(* Logix 5000 project; controller DispersionPlc vendor 1 type 14 code 108 rev 34.11; software revision 34.01; part 6 of 22 *)
(* tags used below, declared in another part *)
   D_AlarmTimers : TIMER[200];
   D_AlarmTimers2 : TIMER[100];
   Disp_AlarmScanIdx : DINT;
   Disp_NewAlarmScanIdx : DINT;
   DispAlarmDisplayTmr : TIMER;
   DispersionAckAlarms : BOOL[128];
   DPT_4320_Holding : REAL;
   DPT_4320_Samples : DINT;
   InxTog : BOOL[32];
   NoNEwAlarmsDestedted : BOOL;
   ONS : BOOL[32];
   _Placeholder : DINT;
   AFB : BOOL;
   AFI : BOOL;
   AG4302_LLP_Alarm : BOOL;
   B4320_PumpAutoCommand : BOOL;
   B4320_PumpManCommand : BOOL;
   B4320_PumpManStart : AOI_Toggle;
   Both_Running : BOOL;
   Both_Running_Timer : TIMER;
   Cat_Destination_K400 : BOOL;
   Cat_Destination_T4301 : BOOL;
   Cat_Tank_Destination : DINT;
   Disp_AlarmsResetting : BOOL;
   Disp_Alr_To_Sound_Horn : BOOL[128];
   Disp_AlrResetIdx : DINT;
   Disp_QuedAlarm : DINT;
   DispAlarmResetBit : BOOL;
   DispersionAlarms : BOOL[256];
   DPT_4320 : REAL;
   DPT_4320_FILL : REAL;
   DPT_4320_Holding1 : REAL;
   DPT_4320_OffSet : REAL;
   DPT_4320_Raw : INT;
   DPT_4320_Sf : REAL;
   dpthighraw : REAL;
   dptlowraw : REAL;
   Drum_Transfer : BOOL;
   Emergency_Cool_4301 : BOOL;
   Enable_High_Alarm : BOOL;
   Estop_Inx : ALIAS FOR Local:3:I.Data.3;
   EstopBulk_upper : ALIAS FOR Local:1:O.Data[27].15;
   FE_4303 : REAL;
   FE_4303_Low : REAL;
   FE_4304 : REAL;
   FE_4304_Low : REAL;
   HMI_Linked_Timer : REAL;
   Hold_For_Flow_Switch : BOOL;
   HornONS_Phases : BOOL[32];
   HS_9A249 : ALIAS FOR Local:1:O.Data[0].17;
   HS_9A640 : ALIAS FOR Local:1:O.Data[0].18;
   InxAlarms : BOOL[128];
   K4_High_Temp : BOOL;
   K4_Low_Temp : BOOL;
   Linked_Timer : TIMER;
   LS_4302_High : BOOL;
   MCC1D4_20_TT5_Relay : BOOL;
   MCC1F3_TT1_Relay : BOOL;
   MCC1F4_8_TT9_Relay : BOOL;
   Melamine_Amount_Per_Count : REAL;
   Melamine_Charge_Remaining : REAL;
   Melamine_Flow_Rate : REAL;
   Melamine_Flow_Raw : INT;
   Melamine_Flow_Raw_Adjusted : REAL;
   Melamine_Flow_Scale_Factor : REAL;
   Melamine_Last_Charge : REAL;
   Melamine_Manual_Start : BOOL;
   Melamine_Pump_Off : BOOL;
   Melamine_Pump_Run : BOOL;
   Melamine_Transfer : BOOL;
   Melamine_transfer_amount : REAL;
   melamine_transfer_setpoint : REAL;
   MelaminePumpTmr : TIMER;
   Melimine_Max_Flow : DINT;
   Melimine_Pump_Manual_Run : BOOL;
   MIXER_A_4320_RUN : ALIAS FOR Local:1:O.Data[0].5;
   MMI_A_4320_RUN_PB : BOOL;
   MMI_Disp_Alarm_Reset_Pb : BOOL;
   MMI_INX_Solvent_Bypass : BOOL;
   MMI_INX_Solvent_Bypass_TOG : BOOL;
   MMI_P_4303_Run_Pb : BOOL;
   MMI_P_4304_RUN_PB : BOOL;
   MMI_P_4320_RUN_PB : BOOL;
   MMI_XV_4320_1_PB : BOOL;
   MMI_XV_4320_2_PB : BOOL;
   Mon_Destination_K400 : BOOL;
   Mon_Destination_T4301 : BOOL;
   Mon_Tank_Destination : DINT;
   NM_4303_AOI : AStd_AI_AOI;
   NM_4303_O2 : AStd_AnalogInput;
   O7_10_BUZ : ALIAS FOR Local:7:O.Data.10;
   One_Shots : DINT;
   OneShots : DINT;
   ONSTog : DINT;
   Phase_AlarmHorn : BOOL;
   Pv_Disp_Alarm_Val : DINT;
   RG_T52_AI_Raw : INT;
   RG_T53_AI_Raw : INT;
   RTA_Input_Floats : REAL[100];
   SPARE_I_1_4_5 : ALIAS FOR Local:1:I.Data[4].5;
   SPARE_O_1_0_21 : ALIAS FOR Local:1:O.Data[0].21;
   ST_K400_1 : REAL;
   ST_K400_1_LOW : REAL;
   ST_K400_1_Timer : TIMER[6];
   ST_K400_SAFETY : BOOL;
   Start_Melamine_Transfer_PB : BOOL;
   T4301_AIR_PURGE_REQUEST : BOOL;
   T4301_Cooling_On : BOOL;
   T4301_Heating_On : BOOL;
   T4301_K : Kettle;
   T4301_Mixer : VFD;
   T4301_Process_Alarm_Setpoints : Alarm_SPT;
   T4301_Temp_Feed_Alarm : DINT;
   T4302_Cooling_Pressure : DINT;
   T4302_Cooling_Pressure_SPT : DINT;
   T4302_DISCHARGE : BOOL;
   t4302_Line_pressure_High : BOOL;
   t4302_Line_pressure_Hightmr : TIMER;
   T53_Mixer : VFD;
   Tank_Link_Enable : BOOL;
   Tank_Link_Enable_ONS : BOOL;
   Tank_Link_Enable_ONS1 : BOOL;
   Tank_Link_ONS : BOOL[32];
   Tank_Linked : BOOL;
   TE_4301A : ALIAS FOR Local:8:I.Ch0Data;
   Te_4301A_High : REAL;
   TE_4301A_Low : REAL;
   TE_4320 : INT;
   TIT_S51_1 : AStd_AnalogInput;
   TOGGLE : BOOL;
   TRANS_PUMP_P_4320_RUN : ALIAS FOR Local:1:O.Data[0].6;
   TransferDone : BOOL;
   TruckLoadLevelAlarmResetPBLight : BOOL;
   V4304_Pump : VFD;
   Vaild_Monomer_Barcode : BOOL;
   VFD_4302_1 : AStd_VFD;
   W4303_Pump : VFD;
   WIT_4302_1 : AStd_AnalogInput;
   WIT_4306_1 : AStd_AnalogInput;
   WIT_4307_1 : AStd_AnalogInput;
   XI_K400_1 : BOOL;
   XV_4303_01 : ALIAS FOR Local:5:O.Data.3;
   XV_4303_03 : BOOL;
   XV_4303_04 : BOOL;
   XV_4303_05 : BOOL;
   XV_4304 : ALIAS FOR Local:5:O.Data.4;
   XV_4304_02 : BOOL;
   XV_4304_03 : BOOL;
   XV_4304_04 : BOOL;
   XV_4320_1 : ALIAS FOR Local:1:O.Data[1].1;
   XV_4320_2 : ALIAS FOR Local:1:O.Data[1].0;
   XV_K400_03_SEQCLOSE : BOOL;
   XV_K400_04_SEQCLOSE : BOOL;
   ZSC_4303_03 : BOOL;
   ZSC_4303_04 : BOOL;
   ZSC_4303_05 : BOOL;
   ZSC_4304_02 : BOOL;
   ZSC_4304_03 : BOOL;
   ZSC_4304_04 : BOOL;
   ZSC_4320_1 : ALIAS FOR Local:1:I.Data[4].3;
   ZSO_4303_03 : BOOL;
   ZSO_4303_04 : BOOL;
   ZSO_4303_05 : BOOL;
   ZSO_4304_02 : BOOL;
   ZSO_4304_03 : BOOL;
   ZSO_4304_04 : BOOL;
   ZSO_4320_1 : ALIAS FOR Local:1:I.Data[4].2;
   ZSO_4320_2 : ALIAS FOR Local:1:I.Data[4].0;
(* MainProgram, continued *)

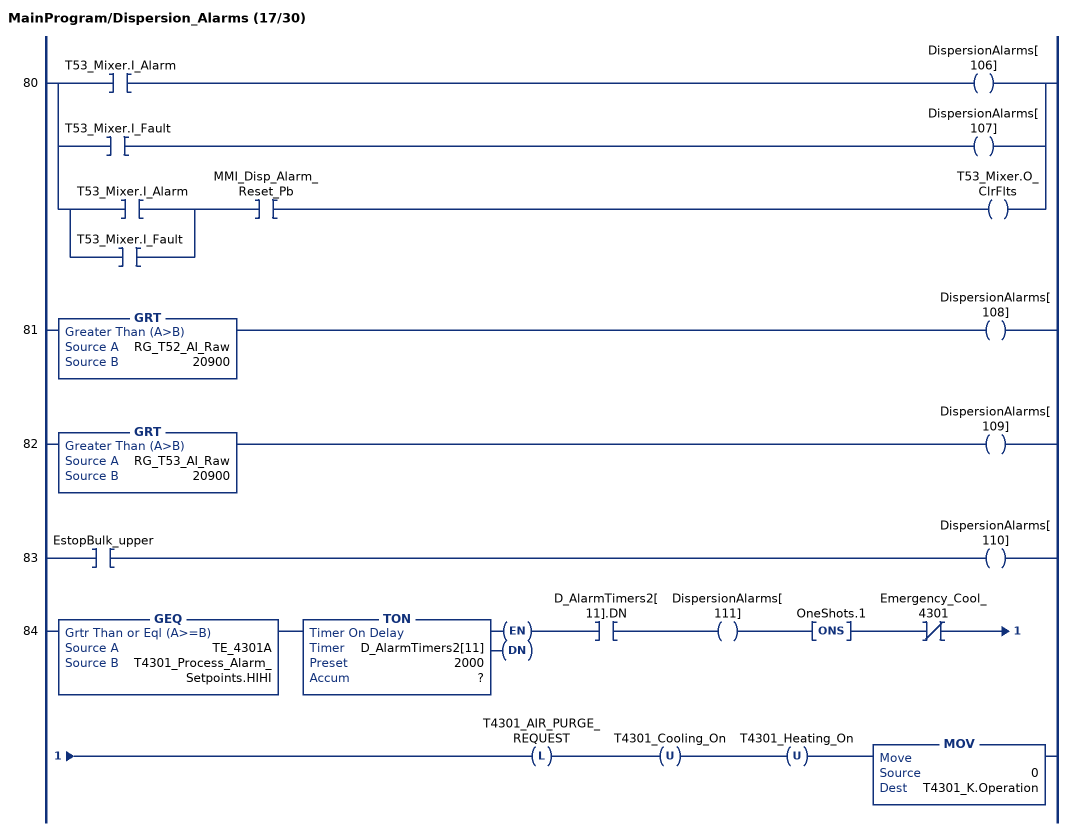
   [picture p93: MainProgram/Dispersion_Alarms rungs 80-84]
   80: [XIC(T53_Mixer.I_Alarm) OTE(DispersionAlarms[106]) ,XIC(T53_Mixer.I_Fault) OTE(DispersionAlarms[107]) ,[XIC(T53_Mixer.I_Alarm) ,XIC(T53_Mixer.I_Fault) ] XIC(MMI_Disp_Alarm_Reset_Pb) OTE(T53_Mixer.O_ClrFlts) ];
   81: GRT(RG_T52_AI_Raw,20900)OTE(DispersionAlarms[108]);
   82: GRT(RG_T53_AI_Raw,20900)OTE(DispersionAlarms[109]);
   83: XIC(EstopBulk_upper)OTE(DispersionAlarms[110]);
   84: GEQ(TE_4301A,T4301_Process_Alarm_Setpoints.HIHI)TON(D_AlarmTimers2[11],?,?)XIC(D_AlarmTimers2[11].DN)OTE(DispersionAlarms[111])ONS(OneShots.1)XIO(Emergency_Cool_4301)OTL(T4301_AIR_PURGE_REQUEST)OTU(T4301_Cooling_On)OTU(T4301_Heating_On)MOV(0,T4301_K.Operation);
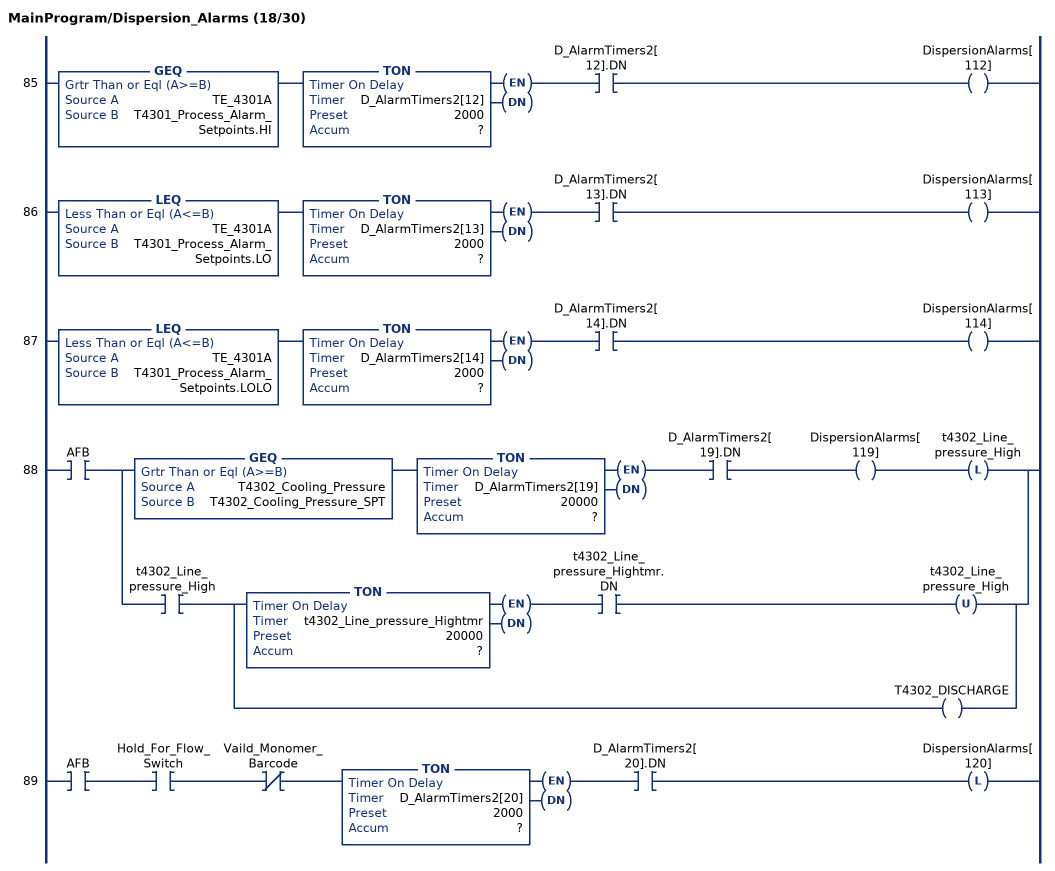
   85: GEQ(TE_4301A,T4301_Process_Alarm_Setpoints.HI)TON(D_AlarmTimers2[12],?,?)XIC(D_AlarmTimers2[12].DN)OTE(DispersionAlarms[112]);
   86: LEQ(TE_4301A,T4301_Process_Alarm_Setpoints.LO)TON(D_AlarmTimers2[13],?,?)XIC(D_AlarmTimers2[13].DN)OTE(DispersionAlarms[113]);
   87: LEQ(TE_4301A,T4301_Process_Alarm_Setpoints.LOLO)TON(D_AlarmTimers2[14],?,?)XIC(D_AlarmTimers2[14].DN)OTE(DispersionAlarms[114]);
   88: XIC(AFB)[GEQ(T4302_Cooling_Pressure,T4302_Cooling_Pressure_SPT) TON(D_AlarmTimers2[19],?,?) XIC(D_AlarmTimers2[19].DN) OTE(DispersionAlarms[119]) OTL(t4302_Line_pressure_High) ,XIC(t4302_Line_pressure_High) [TON(t4302_Line_pressure_Hightmr,?,?) XIC(t4302_Line_pressure_Hightmr.DN) OTU(t4302_Line_pressure_High) ,OTE(T4302_DISCHARGE) ] ];
   89: XIC(AFB)XIC(Hold_For_Flow_Switch)XIO(Vaild_Monomer_Barcode)TON(D_AlarmTimers2[20],?,?)XIC(D_AlarmTimers2[20].DN)OTL(DispersionAlarms[120]);
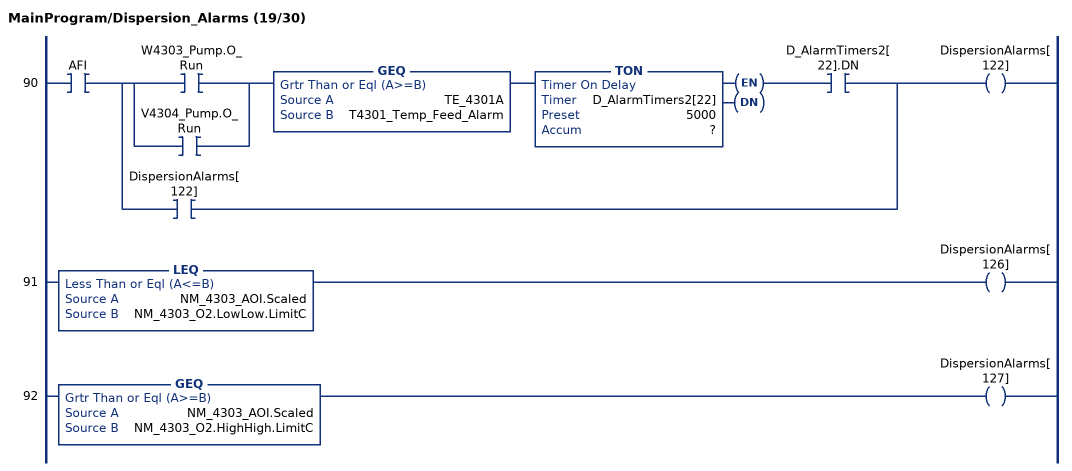
   90: XIC(AFI)[[XIC(W4303_Pump.O_Run) ,XIC(V4304_Pump.O_Run) ] GEQ(TE_4301A,T4301_Temp_Feed_Alarm) TON(D_AlarmTimers2[22],?,?) XIC(D_AlarmTimers2[22].DN) ,XIC(DispersionAlarms[122]) ]OTE(DispersionAlarms[122]);
   91: LEQ(NM_4303_AOI.Scaled,NM_4303_O2.LowLow.LimitC)OTE(DispersionAlarms[126]);
   92: GEQ(NM_4303_AOI.Scaled,NM_4303_O2.HighHigh.LimitC)OTE(DispersionAlarms[127]);
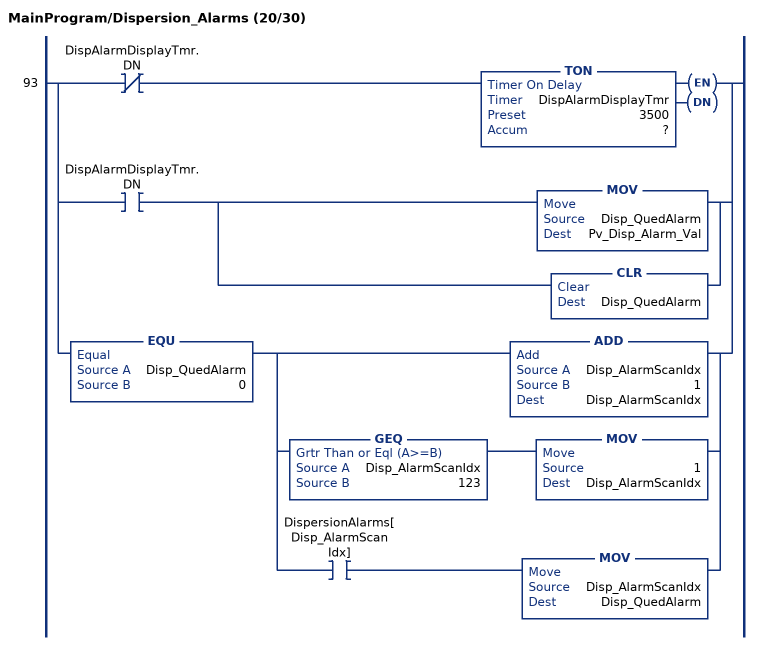
   93: [XIO(DispAlarmDisplayTmr.DN) TON(DispAlarmDisplayTmr,?,?) ,XIC(DispAlarmDisplayTmr.DN) [MOV(Disp_QuedAlarm,Pv_Disp_Alarm_Val) ,CLR(Disp_QuedAlarm) ] ,EQU(Disp_QuedAlarm,0) [ADD(Disp_AlarmScanIdx,1,Disp_AlarmScanIdx) ,GEQ(Disp_AlarmScanIdx,123) MOV(1,Disp_AlarmScanIdx) ,XIC(DispersionAlarms[Disp_AlarmScanIdx]) MOV(Disp_AlarmScanIdx,Disp_QuedAlarm) ] ];
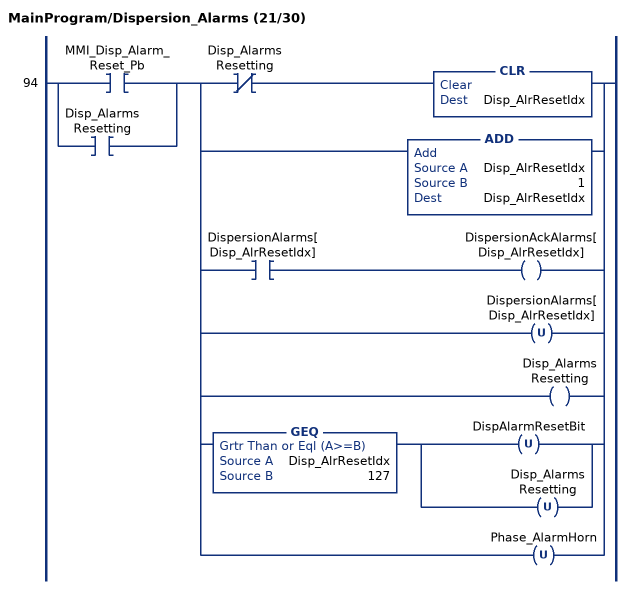
   94: [XIC(MMI_Disp_Alarm_Reset_Pb) ,XIC(Disp_AlarmsResetting) ][XIO(Disp_AlarmsResetting) CLR(Disp_AlrResetIdx) ,ADD(Disp_AlrResetIdx,1,Disp_AlrResetIdx) ,XIC(DispersionAlarms[Disp_AlrResetIdx]) OTE(DispersionAckAlarms[Disp_AlrResetIdx]) ,OTU(DispersionAlarms[Disp_AlrResetIdx]) ,OTE(Disp_AlarmsResetting) ,GEQ(Disp_AlrResetIdx,127) [OTU(DispAlarmResetBit) ,OTU(Disp_AlarmsResetting) ] ,OTU(Phase_AlarmHorn) ];
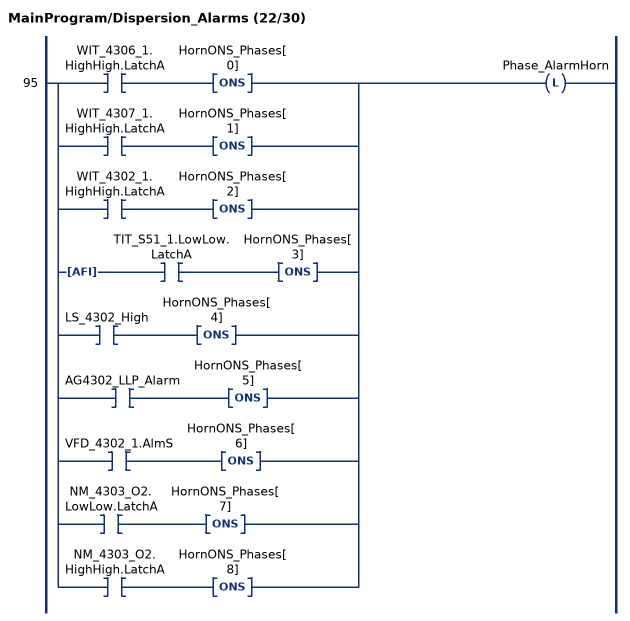
   95: [XIC(WIT_4306_1.HighHigh.LatchA) ONS(HornONS_Phases[0]) ,XIC(WIT_4307_1.HighHigh.LatchA) ONS(HornONS_Phases[1]) ,XIC(WIT_4302_1.HighHigh.LatchA) ONS(HornONS_Phases[2]) ,AFI() XIC(TIT_S51_1.LowLow.LatchA) ONS(HornONS_Phases[3]) ,XIC(LS_4302_High) ONS(HornONS_Phases[4]) ,XIC(AG4302_LLP_Alarm) ONS(HornONS_Phases[5]) ,XIC(VFD_4302_1.AlmS) ONS(HornONS_Phases[6]) ,XIC(NM_4303_O2.LowLow.LatchA) ONS(HornONS_Phases[7]) ,XIC(NM_4303_O2.HighHigh.LatchA) ONS(HornONS_Phases[8]) ]OTL(Phase_AlarmHorn);
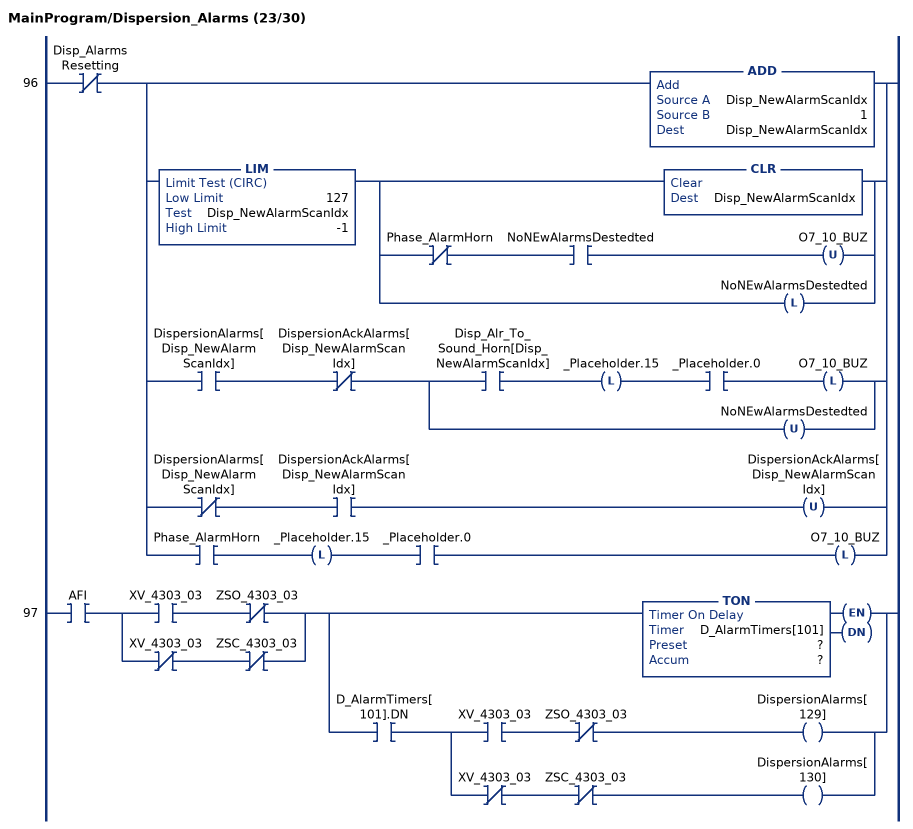
   96: XIO(Disp_AlarmsResetting)[ADD(Disp_NewAlarmScanIdx,1,Disp_NewAlarmScanIdx) ,LIM(127,Disp_NewAlarmScanIdx,-1) [CLR(Disp_NewAlarmScanIdx) ,XIO(Phase_AlarmHorn) XIC(NoNEwAlarmsDestedted) OTU(O7_10_BUZ) ,OTL(NoNEwAlarmsDestedted) ] ,XIC(DispersionAlarms[Disp_NewAlarmScanIdx]) XIO(DispersionAckAlarms[Disp_NewAlarmScanIdx]) [XIC(Disp_Alr_To_Sound_Horn[Disp_NewAlarmScanIdx]) OTL(_Placeholder.15) XIC(_Placeholder.0) OTL(O7_10_BUZ) ,OTU(NoNEwAlarmsDestedted) ] ,XIO(DispersionAlarms[Disp_NewAlarmScanIdx]) XIC(DispersionAckAlarms[Disp_NewAlarmScanIdx]) OTU(DispersionAckAlarms[Disp_NewAlarmScanIdx]) ,XIC(Phase_AlarmHorn) OTL(_Placeholder.15) XIC(_Placeholder.0) OTL(O7_10_BUZ) ];
   97: XIC(AFI)[XIC(XV_4303_03) XIO(ZSO_4303_03) ,XIO(XV_4303_03) XIO(ZSC_4303_03) ][TON(D_AlarmTimers[101],?,?) ,XIC(D_AlarmTimers[101].DN) [XIC(XV_4303_03) XIO(ZSO_4303_03) OTE(DispersionAlarms[129]) ,XIO(XV_4303_03) XIO(ZSC_4303_03) OTE(DispersionAlarms[130]) ] ];
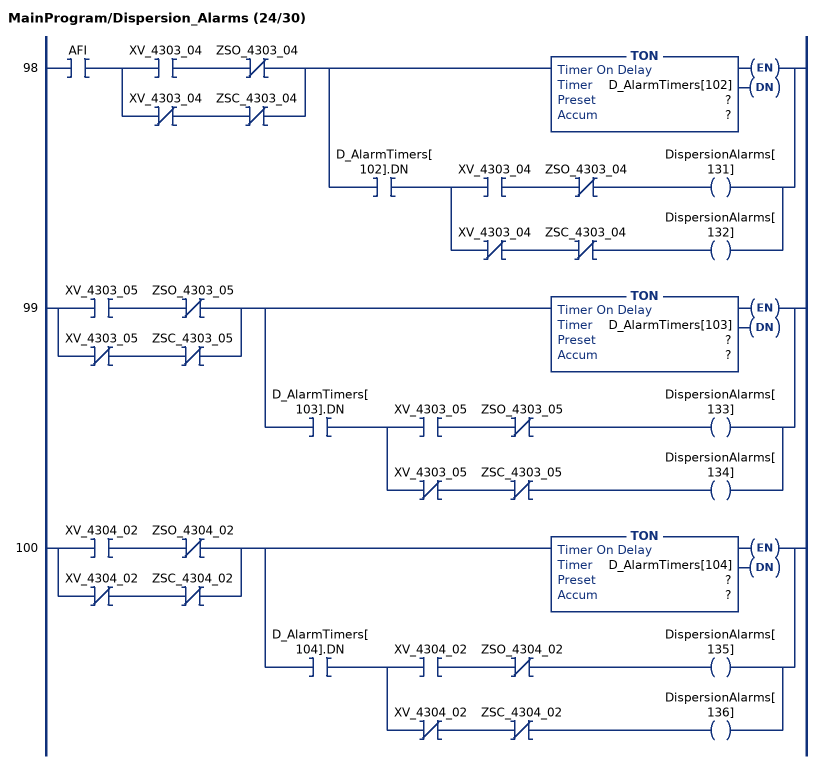
   98: XIC(AFI)[XIC(XV_4303_04) XIO(ZSO_4303_04) ,XIO(XV_4303_04) XIO(ZSC_4303_04) ][TON(D_AlarmTimers[102],?,?) ,XIC(D_AlarmTimers[102].DN) [XIC(XV_4303_04) XIO(ZSO_4303_04) OTE(DispersionAlarms[131]) ,XIO(XV_4303_04) XIO(ZSC_4303_04) OTE(DispersionAlarms[132]) ] ];
   99: [XIC(XV_4303_05) XIO(ZSO_4303_05) ,XIO(XV_4303_05) XIO(ZSC_4303_05) ][TON(D_AlarmTimers[103],?,?) ,XIC(D_AlarmTimers[103].DN) [XIC(XV_4303_05) XIO(ZSO_4303_05) OTE(DispersionAlarms[133]) ,XIO(XV_4303_05) XIO(ZSC_4303_05) OTE(DispersionAlarms[134]) ] ];
   100: [XIC(XV_4304_02) XIO(ZSO_4304_02) ,XIO(XV_4304_02) XIO(ZSC_4304_02) ][TON(D_AlarmTimers[104],?,?) ,XIC(D_AlarmTimers[104].DN) [XIC(XV_4304_02) XIO(ZSO_4304_02) OTE(DispersionAlarms[135]) ,XIO(XV_4304_02) XIO(ZSC_4304_02) OTE(DispersionAlarms[136]) ] ];
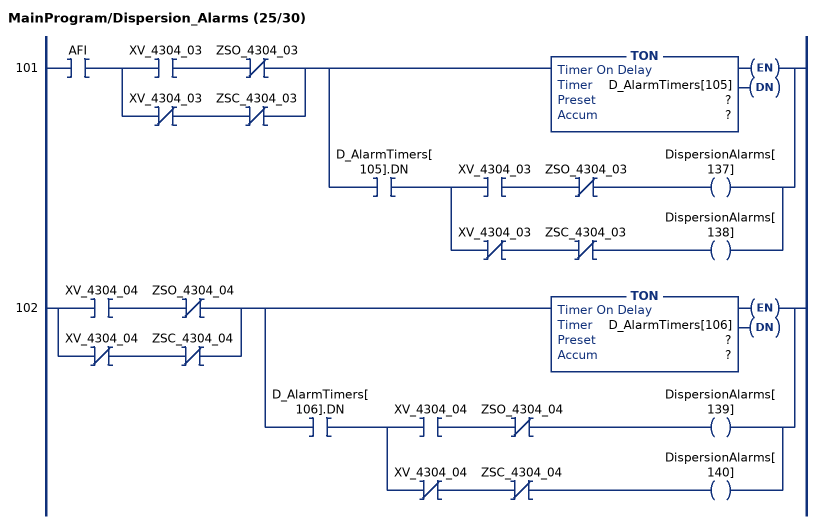
   101: XIC(AFI)[XIC(XV_4304_03) XIO(ZSO_4304_03) ,XIO(XV_4304_03) XIO(ZSC_4304_03) ][TON(D_AlarmTimers[105],?,?) ,XIC(D_AlarmTimers[105].DN) [XIC(XV_4304_03) XIO(ZSO_4304_03) OTE(DispersionAlarms[137]) ,XIO(XV_4304_03) XIO(ZSC_4304_03) OTE(DispersionAlarms[138]) ] ];
   102: [XIC(XV_4304_04) XIO(ZSO_4304_04) ,XIO(XV_4304_04) XIO(ZSC_4304_04) ][TON(D_AlarmTimers[106],?,?) ,XIC(D_AlarmTimers[106].DN) [XIC(XV_4304_04) XIO(ZSO_4304_04) OTE(DispersionAlarms[139]) ,XIO(XV_4304_04) XIO(ZSC_4304_04) OTE(DispersionAlarms[140]) ] ];
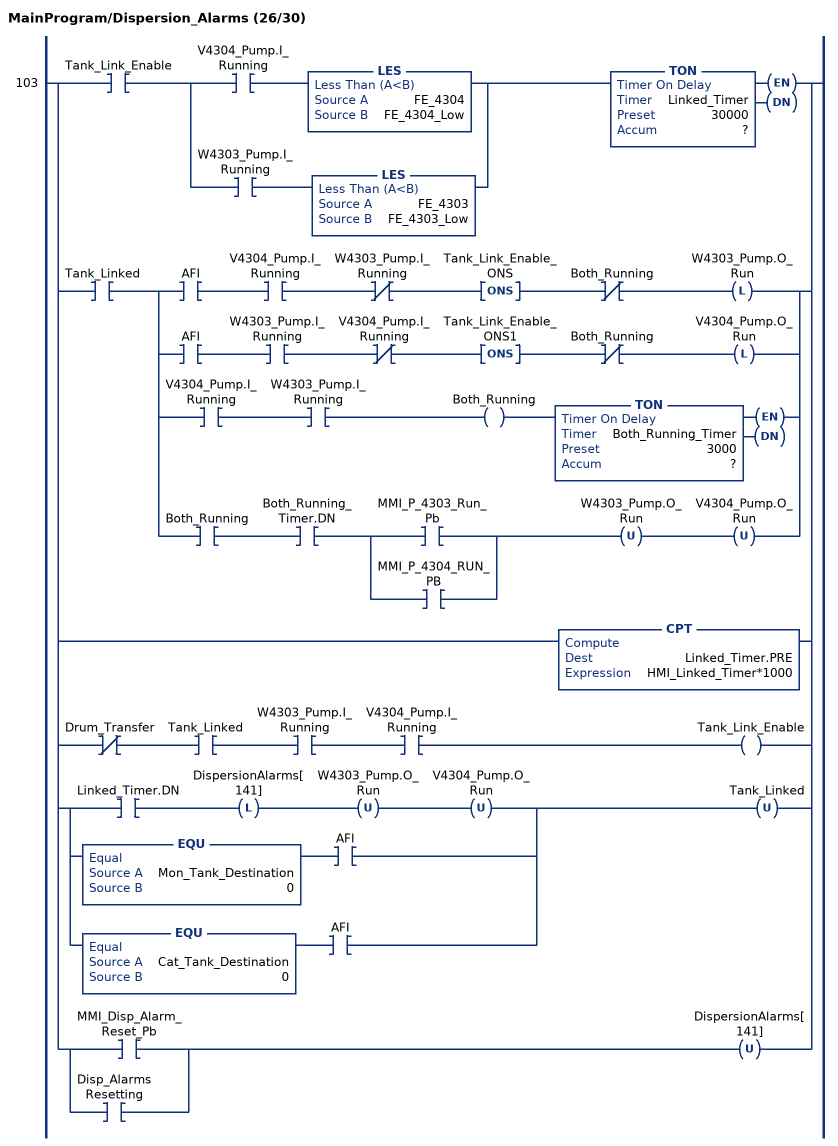
   103: [XIC(Tank_Link_Enable) [XIC(V4304_Pump.I_Running) LES(FE_4304,FE_4304_Low) ,XIC(W4303_Pump.I_Running) LES(FE_4303,FE_4303_Low) ] TON(Linked_Timer,?,?) ,XIC(Tank_Linked) [XIC(AFI) XIC(V4304_Pump.I_Running) XIO(W4303_Pump.I_Running) ONS(Tank_Link_Enable_ONS) XIO(Both_Running) OTL(W4303_Pump.O_Run) ,XIC(AFI) XIC(W4303_Pump.I_Running) XIO(V4304_Pump.I_Running) ONS(Tank_Link_Enable_ONS1) XIO(Both_Running) OTL(V4304_Pump.O_Run) ,XIC(V4304_Pump.I_Running) XIC(W4303_Pump.I_Running) OTE(Both_Running) TON(Both_Running_Timer,?,?) ,XIC(Both_Running) XIC(Both_Running_Timer.DN) [XIC(MMI_P_4303_Run_Pb) ,XIC(MMI_P_4304_RUN_PB) ] OTU(W4303_Pump.O_Run) OTU(V4304_Pump.O_Run) ] ,CPT(Linked_Timer.PRE,HMI_Linked_Timer*1000) ,XIO(Drum_Transfer) XIC(Tank_Linked) XIC(W4303_Pump.I_Running) XIC(V4304_Pump.I_Running) OTE(Tank_Link_Enable) ,[XIC(Linked_Timer.DN) OTL(DispersionAlarms[141]) OTU(W4303_Pump.O_Run) OTU(V4304_Pump.O_Run) ,EQU(Mon_Tank_Destination,0) XIC(AFI) ,EQU(Cat_Tank_Destination,0) XIC(AFI) ] OTU(Tank_Linked) ,[XIC(MMI_Disp_Alarm_Reset_Pb) ,XIC(Disp_AlarmsResetting) ] OTU(DispersionAlarms[141]) ];
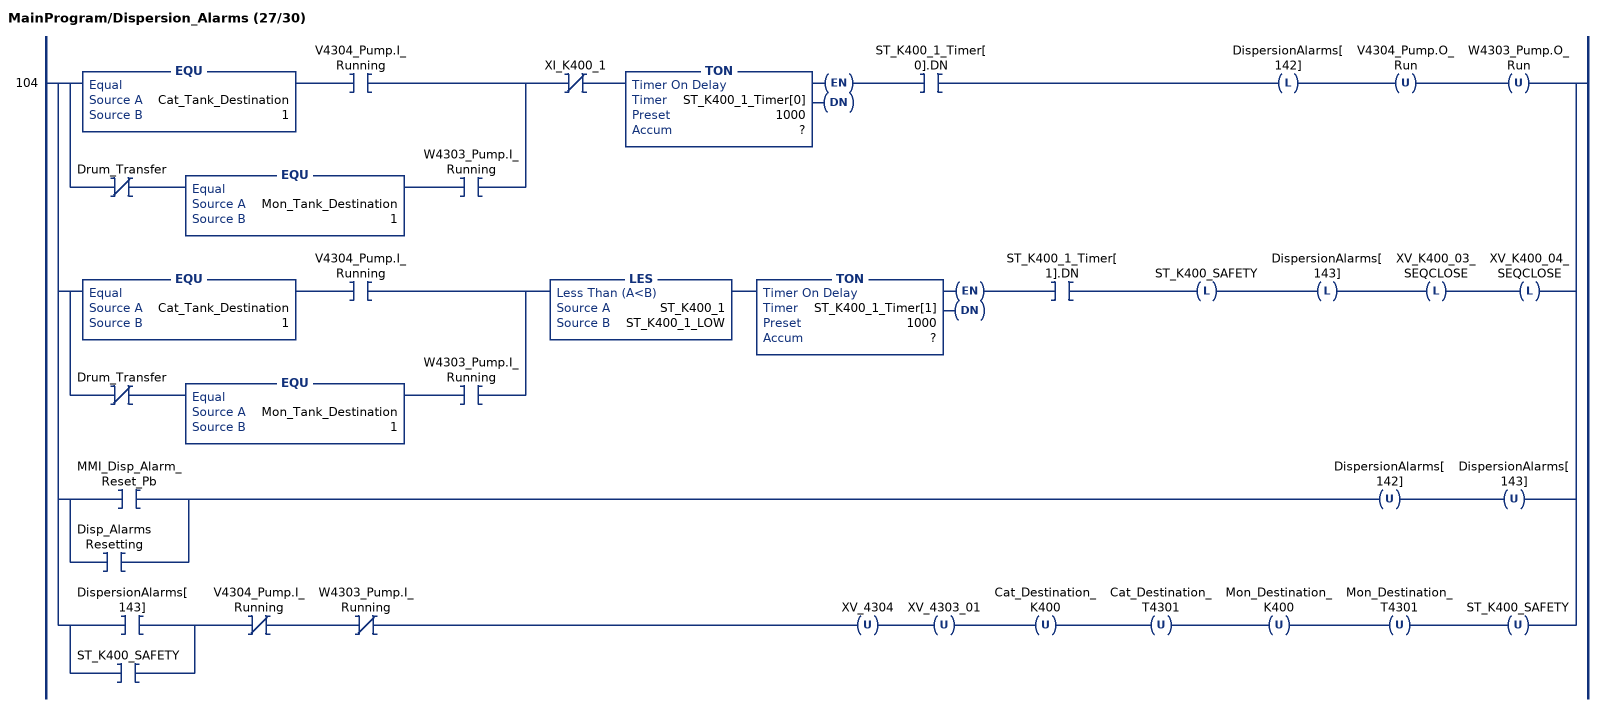
   104: [[EQU(Cat_Tank_Destination,1) XIC(V4304_Pump.I_Running) ,XIO(Drum_Transfer) EQU(Mon_Tank_Destination,1) XIC(W4303_Pump.I_Running) ] XIO(XI_K400_1) TON(ST_K400_1_Timer[0],?,?) XIC(ST_K400_1_Timer[0].DN) OTL(DispersionAlarms[142]) OTU(V4304_Pump.O_Run) OTU(W4303_Pump.O_Run) ,[EQU(Cat_Tank_Destination,1) XIC(V4304_Pump.I_Running) ,XIO(Drum_Transfer) EQU(Mon_Tank_Destination,1) XIC(W4303_Pump.I_Running) ] LES(ST_K400_1,ST_K400_1_LOW) TON(ST_K400_1_Timer[1],?,?) XIC(ST_K400_1_Timer[1].DN) OTL(ST_K400_SAFETY) OTL(DispersionAlarms[143]) OTL(XV_K400_03_SEQCLOSE) OTL(XV_K400_04_SEQCLOSE) ,[XIC(MMI_Disp_Alarm_Reset_Pb) ,XIC(Disp_AlarmsResetting) ] OTU(DispersionAlarms[142]) OTU(DispersionAlarms[143]) ,[XIC(DispersionAlarms[143]) ,XIC(ST_K400_SAFETY) ] XIO(V4304_Pump.I_Running) XIO(W4303_Pump.I_Running) OTU(XV_4304) OTU(XV_4303_01) OTU(Cat_Destination_K400) OTU(Cat_Destination_T4301) OTU(Mon_Destination_K400) OTU(Mon_Destination_T4301) OTU(ST_K400_SAFETY) ];
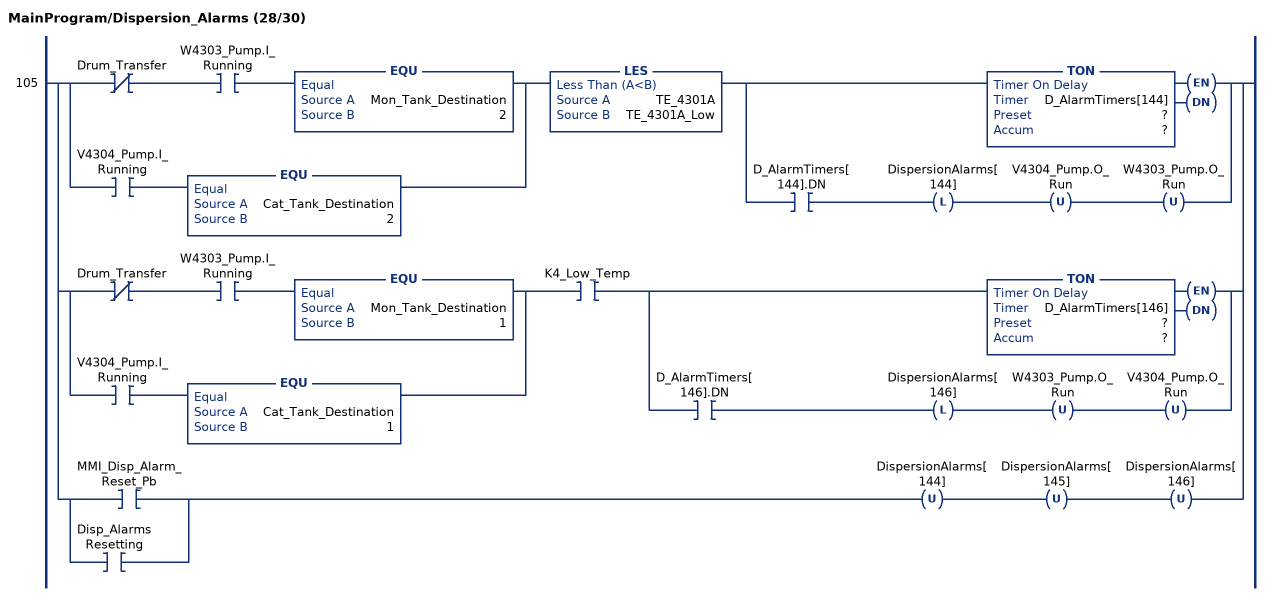
   105: [[[XIO(Drum_Transfer) XIC(W4303_Pump.I_Running) EQU(Mon_Tank_Destination,2) ,XIC(V4304_Pump.I_Running) EQU(Cat_Tank_Destination,2) ] LES(TE_4301A,TE_4301A_Low) [TON(D_AlarmTimers[144],?,?) ,XIC(D_AlarmTimers[144].DN) OTL(DispersionAlarms[144]) OTU(V4304_Pump.O_Run) OTU(W4303_Pump.O_Run) ] ,[XIO(Drum_Transfer) XIC(W4303_Pump.I_Running) EQU(Mon_Tank_Destination,1) ,XIC(V4304_Pump.I_Running) EQU(Cat_Tank_Destination,1) ] XIC(K4_Low_Temp) [TON(D_AlarmTimers[146],?,?) ,XIC(D_AlarmTimers[146].DN) OTL(DispersionAlarms[146]) OTU(W4303_Pump.O_Run) OTU(V4304_Pump.O_Run) ] ] ,[XIC(MMI_Disp_Alarm_Reset_Pb) ,XIC(Disp_AlarmsResetting) ] OTU(DispersionAlarms[144]) OTU(DispersionAlarms[145]) OTU(DispersionAlarms[146]) ];
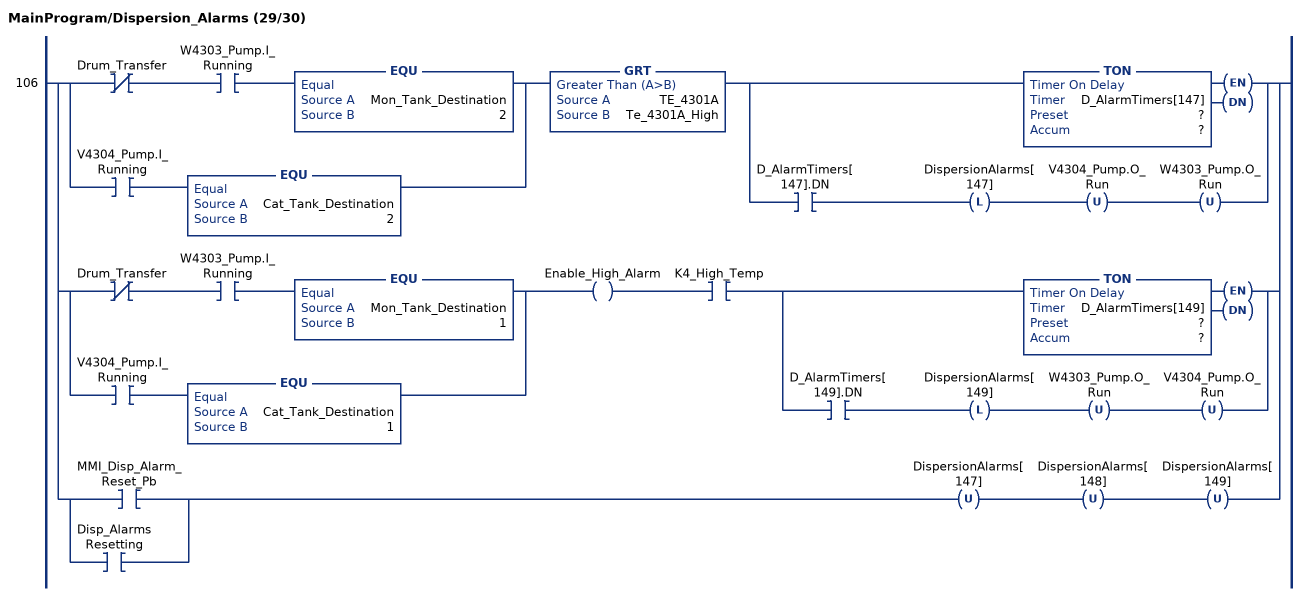
   106: [[[XIO(Drum_Transfer) XIC(W4303_Pump.I_Running) EQU(Mon_Tank_Destination,2) ,XIC(V4304_Pump.I_Running) EQU(Cat_Tank_Destination,2) ] GRT(TE_4301A,Te_4301A_High) [TON(D_AlarmTimers[147],?,?) ,XIC(D_AlarmTimers[147].DN) OTL(DispersionAlarms[147]) OTU(V4304_Pump.O_Run) OTU(W4303_Pump.O_Run) ] ,[XIO(Drum_Transfer) XIC(W4303_Pump.I_Running) EQU(Mon_Tank_Destination,1) ,XIC(V4304_Pump.I_Running) EQU(Cat_Tank_Destination,1) ] OTE(Enable_High_Alarm) XIC(K4_High_Temp) [TON(D_AlarmTimers[149],?,?) ,XIC(D_AlarmTimers[149].DN) OTL(DispersionAlarms[149]) OTU(W4303_Pump.O_Run) OTU(V4304_Pump.O_Run) ] ] ,[XIC(MMI_Disp_Alarm_Reset_Pb) ,XIC(Disp_AlarmsResetting) ] OTU(DispersionAlarms[147]) OTU(DispersionAlarms[148]) OTU(DispersionAlarms[149]) ];
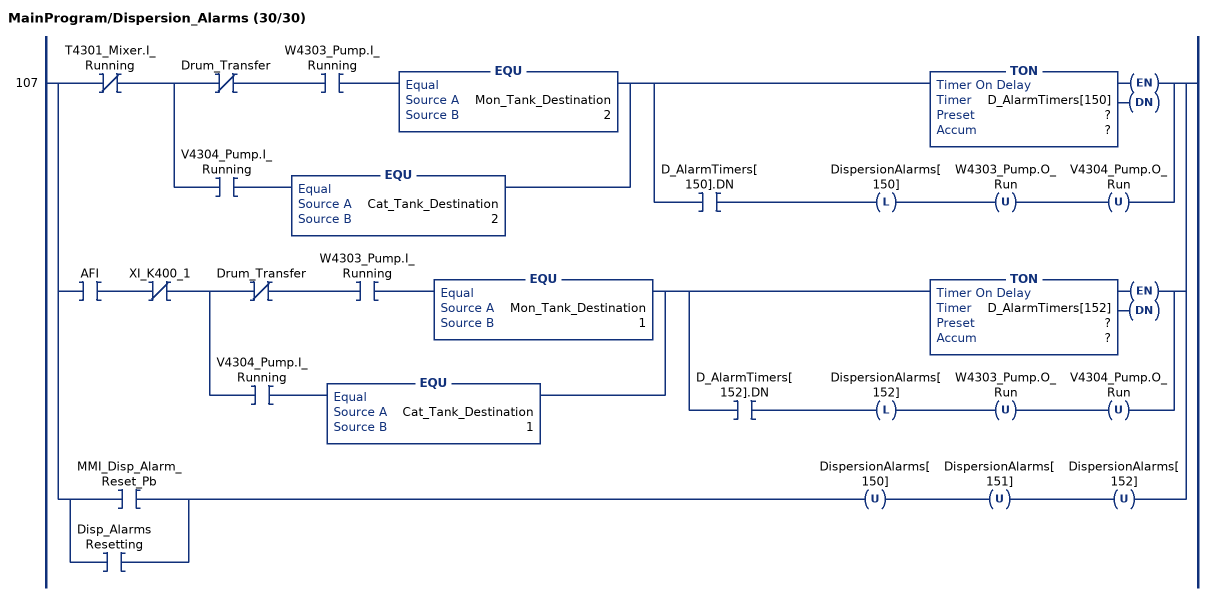
   107: [[XIO(T4301_Mixer.I_Running) [XIO(Drum_Transfer) XIC(W4303_Pump.I_Running) EQU(Mon_Tank_Destination,2) ,XIC(V4304_Pump.I_Running) EQU(Cat_Tank_Destination,2) ] [TON(D_AlarmTimers[150],?,?) ,XIC(D_AlarmTimers[150].DN) OTL(DispersionAlarms[150]) OTU(W4303_Pump.O_Run) OTU(V4304_Pump.O_Run) ] ,XIC(AFI) XIO(XI_K400_1) [XIO(Drum_Transfer) XIC(W4303_Pump.I_Running) EQU(Mon_Tank_Destination,1) ,XIC(V4304_Pump.I_Running) EQU(Cat_Tank_Destination,1) ] [TON(D_AlarmTimers[152],?,?) ,XIC(D_AlarmTimers[152].DN) OTL(DispersionAlarms[152]) OTU(W4303_Pump.O_Run) OTU(V4304_Pump.O_Run) ] ] ,[XIC(MMI_Disp_Alarm_Reset_Pb) ,XIC(Disp_AlarmsResetting) ] OTU(DispersionAlarms[150]) OTU(DispersionAlarms[151]) OTU(DispersionAlarms[152]) ];
END_ROUTINE

ROUTINE INX   (* ladder *)
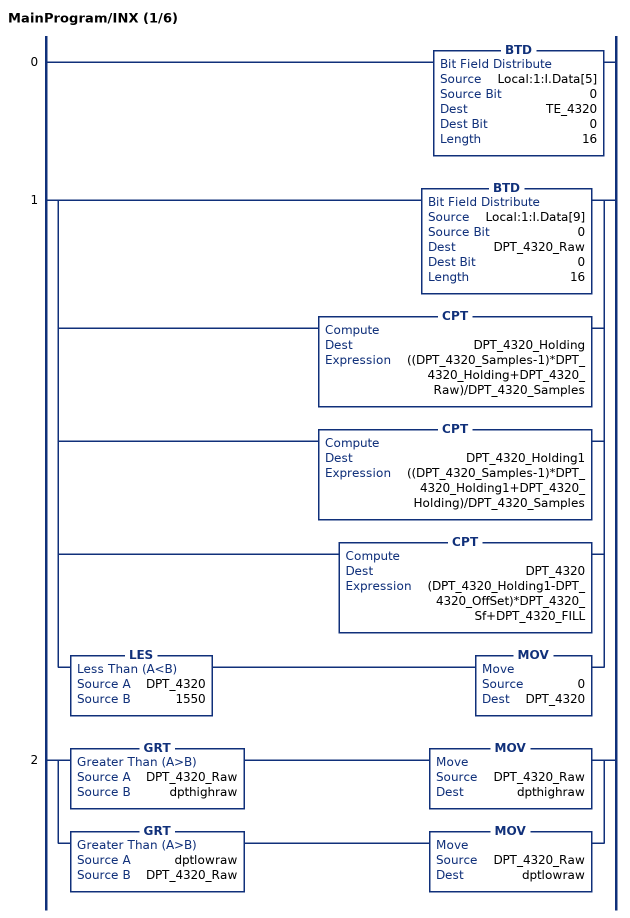
   0: BTD(Local:1:I.Data[5],0,TE_4320,0,16);
   1: [BTD(Local:1:I.Data[9],0,DPT_4320_Raw,0,16) ,CPT(DPT_4320_Holding,((DPT_4320_Samples-1)*DPT_4320_Holding+DPT_4320_Raw)/DPT_4320_Samples) ,CPT(DPT_4320_Holding1,((DPT_4320_Samples-1)*DPT_4320_Holding1+DPT_4320_Holding)/DPT_4320_Samples) ,CPT(DPT_4320,(DPT_4320_Holding1-DPT_4320_OffSet)*DPT_4320_Sf+DPT_4320_FILL) ,LES(DPT_4320,1550) MOV(0,DPT_4320) ];
   2: [GRT(DPT_4320_Raw,dpthighraw) MOV(DPT_4320_Raw,dpthighraw) ,GRT(dptlowraw,DPT_4320_Raw) MOV(DPT_4320_Raw,dptlowraw) ];
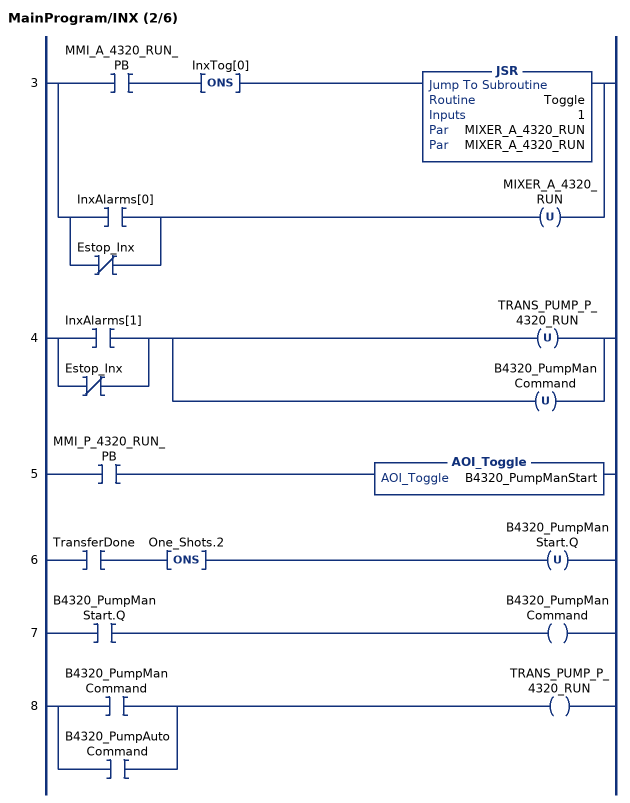
   3: [XIC(MMI_A_4320_RUN_PB) ONS(InxTog[0]) JSR(Toggle,1,MIXER_A_4320_RUN,MIXER_A_4320_RUN) ,[XIC(InxAlarms[0]) ,XIO(Estop_Inx) ] OTU(MIXER_A_4320_RUN) ];
   4: [XIC(InxAlarms[1]) ,XIO(Estop_Inx) ][OTU(TRANS_PUMP_P_4320_RUN) ,OTU(B4320_PumpManCommand) ];
   5: XIC(MMI_P_4320_RUN_PB)AOI_Toggle(B4320_PumpManStart);
   6: XIC(TransferDone)ONS(One_Shots.2)OTU(B4320_PumpManStart.Q);
   7: XIC(B4320_PumpManStart.Q)OTE(B4320_PumpManCommand);
   8: [XIC(B4320_PumpManCommand) ,XIC(B4320_PumpAutoCommand) ]OTE(TRANS_PUMP_P_4320_RUN);
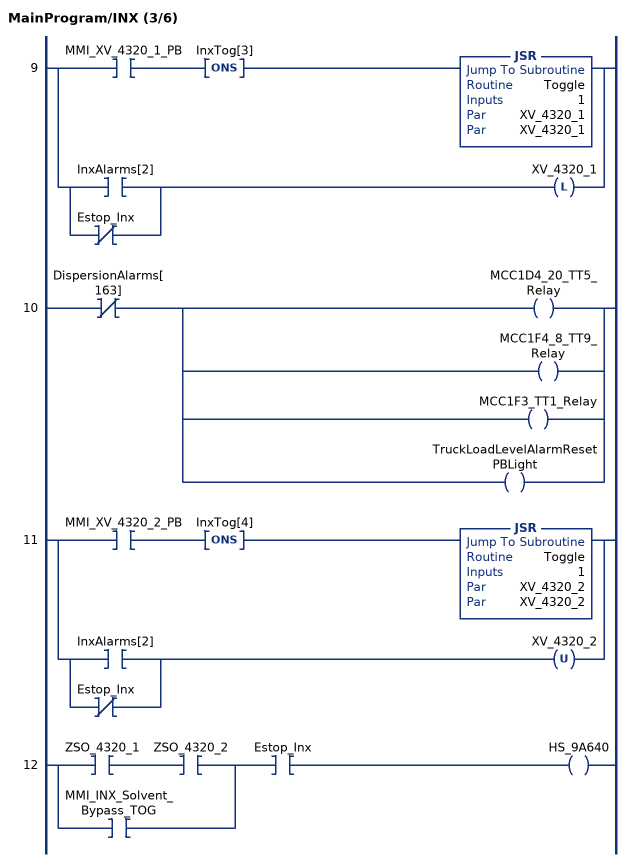
   9: [XIC(MMI_XV_4320_1_PB) ONS(InxTog[3]) JSR(Toggle,1,XV_4320_1,XV_4320_1) ,[XIC(InxAlarms[2]) ,XIO(Estop_Inx) ] OTL(XV_4320_1) ];
   10: XIO(DispersionAlarms[163])[OTE(MCC1D4_20_TT5_Relay) ,OTE(MCC1F4_8_TT9_Relay) ,OTE(MCC1F3_TT1_Relay) ,OTE(TruckLoadLevelAlarmResetPBLight) ];
   11: [XIC(MMI_XV_4320_2_PB) ONS(InxTog[4]) JSR(Toggle,1,XV_4320_2,XV_4320_2) ,[XIC(InxAlarms[2]) ,XIO(Estop_Inx) ] OTU(XV_4320_2) ];
   12: [XIC(ZSO_4320_1) XIC(ZSO_4320_2) ,XIC(MMI_INX_Solvent_Bypass_TOG) ]XIC(Estop_Inx)OTE(HS_9A640);
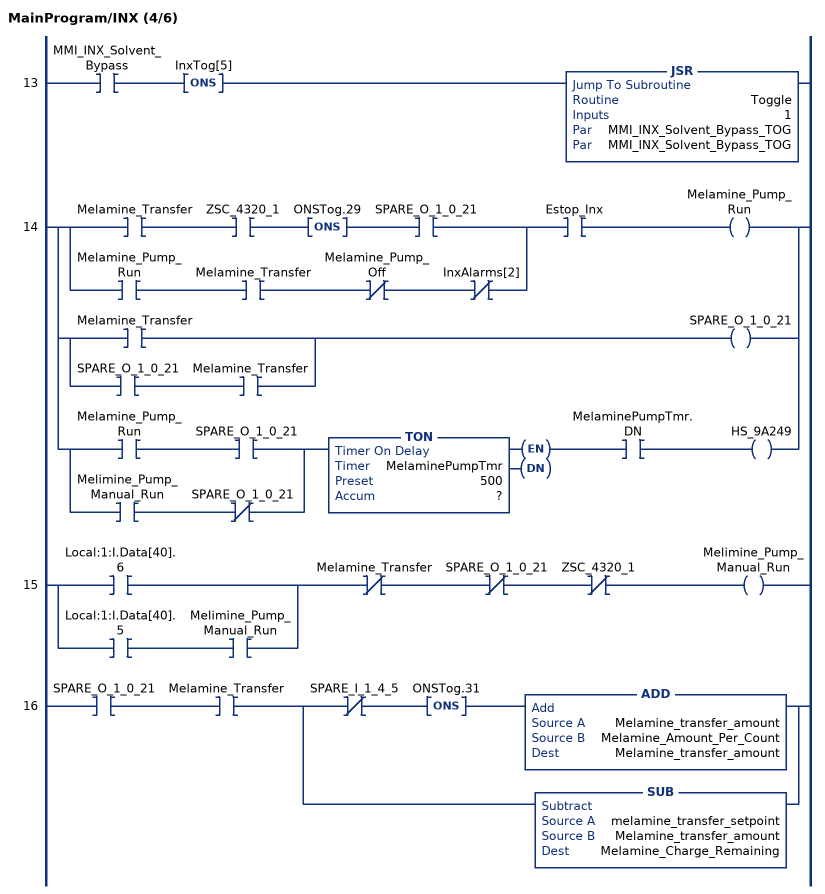
   13: XIC(MMI_INX_Solvent_Bypass)ONS(InxTog[5])JSR(Toggle,1,MMI_INX_Solvent_Bypass_TOG,MMI_INX_Solvent_Bypass_TOG);
   14: [[XIC(Melamine_Transfer) XIC(ZSC_4320_1) ONS(ONSTog.29) XIC(SPARE_O_1_0_21) ,XIC(Melamine_Pump_Run) XIC(Melamine_Transfer) XIO(Melamine_Pump_Off) XIO(InxAlarms[2]) ] XIC(Estop_Inx) OTE(Melamine_Pump_Run) ,[XIC(Melamine_Transfer) ,XIC(SPARE_O_1_0_21) XIC(Melamine_Transfer) ] OTE(SPARE_O_1_0_21) ,[XIC(Melamine_Pump_Run) XIC(SPARE_O_1_0_21) ,XIC(Melimine_Pump_Manual_Run) XIO(SPARE_O_1_0_21) ] TON(MelaminePumpTmr,?,?) XIC(MelaminePumpTmr.DN) OTE(HS_9A249) ];
   15: [XIC(Local:1:I.Data[40].6) ,XIC(Local:1:I.Data[40].5) XIC(Melimine_Pump_Manual_Run) ]XIO(Melamine_Transfer)XIO(SPARE_O_1_0_21)XIO(ZSC_4320_1)OTE(Melimine_Pump_Manual_Run);
   16: XIC(SPARE_O_1_0_21)XIC(Melamine_Transfer)[XIO(SPARE_I_1_4_5) ONS(ONSTog.31) ADD(Melamine_transfer_amount,Melamine_Amount_Per_Count,Melamine_transfer_amount) ,SUB(melamine_transfer_setpoint,Melamine_transfer_amount,Melamine_Charge_Remaining) ];
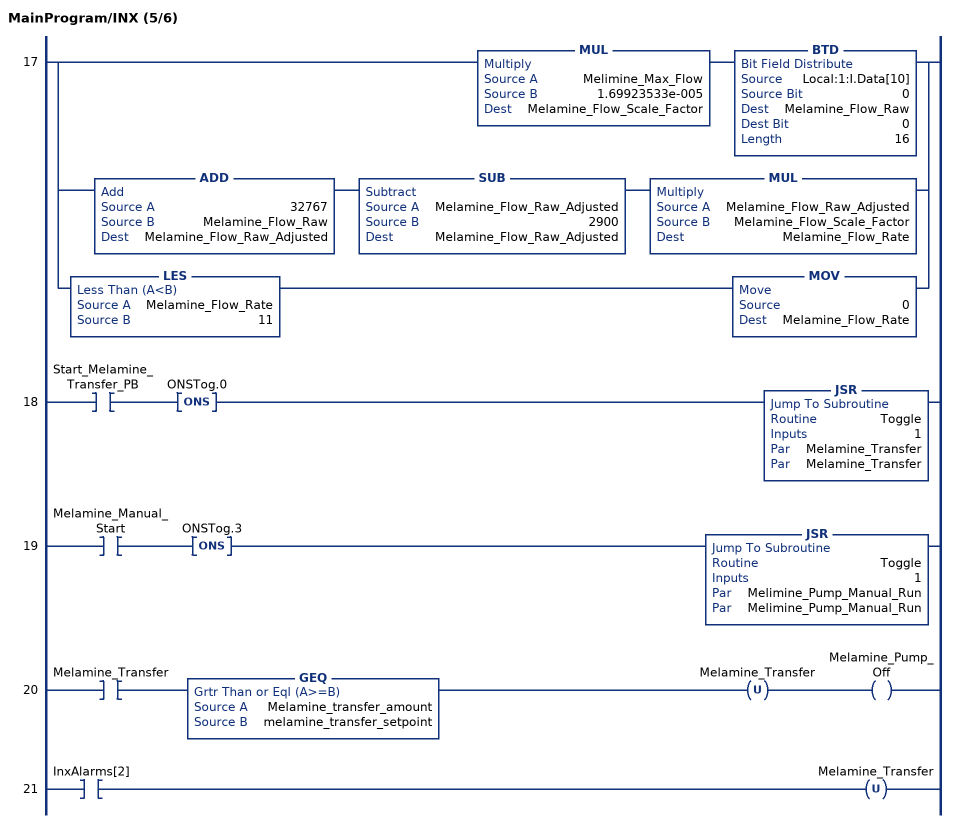
   17: [MUL(Melimine_Max_Flow,1.69923533e-005,Melamine_Flow_Scale_Factor) BTD(Local:1:I.Data[10],0,Melamine_Flow_Raw,0,16) ,ADD(32767,Melamine_Flow_Raw,Melamine_Flow_Raw_Adjusted) SUB(Melamine_Flow_Raw_Adjusted,2900,Melamine_Flow_Raw_Adjusted) MUL(Melamine_Flow_Raw_Adjusted,Melamine_Flow_Scale_Factor,Melamine_Flow_Rate) ,LES(Melamine_Flow_Rate,11) MOV(0,Melamine_Flow_Rate) ];
   18: XIC(Start_Melamine_Transfer_PB)ONS(ONSTog.0)JSR(Toggle,1,Melamine_Transfer,Melamine_Transfer);
   19: XIC(Melamine_Manual_Start)ONS(ONSTog.3)JSR(Toggle,1,Melimine_Pump_Manual_Run,Melimine_Pump_Manual_Run);
   20: XIC(Melamine_Transfer)GEQ(Melamine_transfer_amount,melamine_transfer_setpoint)OTU(Melamine_Transfer)OTE(Melamine_Pump_Off);
   21: XIC(InxAlarms[2])OTU(Melamine_Transfer);
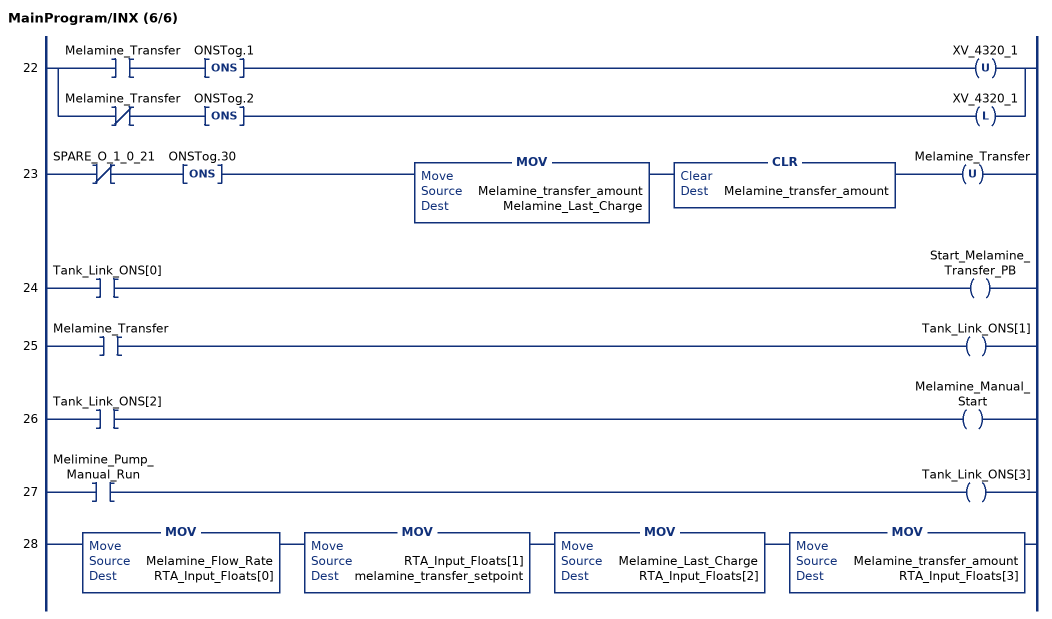
   22: [XIC(Melamine_Transfer) ONS(ONSTog.1) OTU(XV_4320_1) ,XIO(Melamine_Transfer) ONS(ONSTog.2) OTL(XV_4320_1) ];
   23: XIO(SPARE_O_1_0_21)ONS(ONSTog.30)MOV(Melamine_transfer_amount,Melamine_Last_Charge)CLR(Melamine_transfer_amount)OTU(Melamine_Transfer);
   24: XIC(Tank_Link_ONS[0])OTE(Start_Melamine_Transfer_PB);
   25: XIC(Melamine_Transfer)OTE(Tank_Link_ONS[1]);
   26: XIC(Tank_Link_ONS[2])OTE(Melamine_Manual_Start);
   27: XIC(Melimine_Pump_Manual_Run)OTE(Tank_Link_ONS[3]);
   28: MOV(Melamine_Flow_Rate,RTA_Input_Floats[0])MOV(RTA_Input_Floats[1],melamine_transfer_setpoint)MOV(Melamine_Last_Charge,RTA_Input_Floats[2])MOV(Melamine_transfer_amount,RTA_Input_Floats[3]);
END_ROUTINE
